# B&R Automation Studio project automationstudio
Automation Studio 4.9

## Configuration Config1

CPU X20CP1586, AutomationRuntime C4.90, Build 4.1.2, Vc V4.72.2

### Task classes (Cpu.sw)
```
Cyclic#1:
  sensors <- sensors.prg
Cyclic#3:
  main2 <- main2.prg
  main <- main.prg
Binaries: udbdef, FWRules, TCData, sysconf, Role, User, iomap, ashwd, asfw, arconfig, ashwac
Libraries: runtime, astime, asieccon, standard
```

### Hardware
```
X20CP1586 : X20CP1586 v1.8.1.0
  Connector IF2:
    ActivateDevice = 1
  ConfigurationID = sim_assigment_Config1
```

### PvMap.vvm - X20CP1586/PvMap.vvm
```iecst
VAR_CONFIG
	::robot2 AT %Q.::robot2; (*Insert your comment here...*)
	::robot1 AT %Q.::robot1; (*Insert your comment here...*)
END_VAR
```

## Logical view

Binary libraries used (declarations not repeated): standard

### Global.typ - Global data types
```iecst
TYPE
	(* Type with all sensors in scene *)
	sensorsType : STRUCT
		width : ARRAY[0..1] OF INT;
		widthBlocked : ARRAY[0..1] OF BOOL;
		height : ARRAY[0..2] OF INT;
		heightBlocked : ARRAY[0..2] OF BOOL;
		packageForPacker : BOOL;
		packageForPackerPrevious : BOOL;
	END_STRUCT;

	(* Type for holding a set from the package measuring sensors *)
	bufferType : STRUCT
		width : ARRAY[0..1] OF INT;
		height : INT;
	END_STRUCT;

	(* Type with all conveyors in scene *)
	conveyorsType : STRUCT
		circular : conveyorType;			(*  *)
		feed : conveyorType;				(*  *)
		discard : conveyorType;				(*  *)
		packer : conveyorType;				(*  *)
	END_STRUCT;
	(* Type for a specific conveyor *)
	conveyorType : STRUCT
		run : BOOL;			(*  *)
		isOn : BOOL;		(*  *)
	END_STRUCT;

	(* Singular robot control type *)
	robotType : STRUCT
		state : robotStateEnum;		(*  *)
		nextState : robotStateEnum; (*  *)
		target : robotTargetEnum;	(*  *)
		previousTarget : robotTargetEnum; (*  *)
		comm : robotCommunicationType; (*  *)
		grip : BOOL;				(*  *)
		isGripping : BOOL;			(*  *)
		inPosition : BOOL;			(*  *)
		isWaiting : BOOL;			(*  *)
	END_STRUCT;

	(* Robot state Enum *)
	robotStateEnum : (
		RSTATE_INIT, 			(*  *)
		RSTATE_FORCE_HOME,		(*  *)
		RSTATE_WAITING,		(*  *)
		RSTATE_PICKUP,		(*  *)
		RSTATE_PICKUP_R,
		RSTATE_DROP,		(*  *)
		RSTATE_DROP_R,
		RSTATE_CLEAR,
		RSTATE_E_STOP		(*  *)
	);
	(* Robot target/path Enum *)
	robotTargetEnum : (
		RTARGET_FORCE_HOME := 0,	(*  *)
		RTARGET_PICKUP_1 := 10,		(*  *)
		RTARGET_PICKUP_1_R := 11,	(*  *)
		RTARGET_PICKUP_2 := 20,		(*  *)
		RTARGET_PICKUP_2_R := 21,	(*  *)
		RTARGET_PICKUP_3 := 30,		(*  *)
		RTARGET_PICKUP_3_R := 31,	(*  *)
		RTARGET_PICKUP_4 := 40,		(*  *)
		RTARGET_PICKUP_4_R := 41,	(*  *)
		RTARGET_DROPOFF_1 := 50,	(*  *)
		RTARGET_DROPOFF_1_R := 51,	(*  *)
		RTARGET_DROPOFF_2 := 60,	(*  *)
		RTARGET_DROPOFF_2_R := 61,	(*  *)
		RTARGET_DROPOFF_3 := 70,	(*  *)
		RTARGET_DROPOFF_3_R := 71,	(*  *)
		RTARGET_CLEAR := 99			(*  *)
	);

	(*  *)
	sensorStateEnum : (
		STATE_SENSOR_CONVEYOR_INIT := 0,
		STATE_SENSOR_CONVEYOR_STOP := 1,
		STATE_SENSOR_CONVEYOR_START := 2,
		STATE_SENSOR_WAIT,
		STATE_SENSOR_MEASURING,
		STATE_SENSOR_CALCULATING,
		STATE_SENSOR_WAIT_FOR_PICKUP
	);

	(* Type for wrapping single robot comms to RobotStudio Controller *)
	robotCommunicationType : STRUCT
		targets : robotTargetType; (*  *)
		isWaiting : BOOL; (* Is waiting / ready for new action *)
		inPosition : BOOL; (* Is in the last requested position *)
		doGrip : BOOL;	(* Digital output to the gripper *)
		diGrip : BOOL; 	(* Digital input from the gripper *)
	END_STRUCT;

	(*  *)
	robotTargetType : STRUCT
		initHome : BOOL;	(* Communication to the robot *)
		home : BOOL;		(*  happens through booleans  *)
		pick1 : BOOL;		(*  only.                     *)
		pick2 : BOOL;		(* We've not been able to r/w *)
		pick3 : BOOL;		(*  other datatypes.          *)
		pick4 : BOOL;		(* initHome overrides to home *)
		drop1 : BOOL;		(* home with target reverses  *)
		drop2 : BOOL;		(*  the target path.          *)
		drop3 : BOOL;		(*                            *)
	END_STRUCT;

	(* Feeder control type *)
	packFeederType : STRUCT
		doFeed : BOOL;
		isFeeding : BOOL;
	END_STRUCT;

	(* Enum of package sizes *)
	packageSizeEnum :
		(
		PACKAGE_INVALID,
		PACKAGE_SMALL,
		PACKAGE_MEDIUM,
		PACKAGE_LARGE
	);

	(* Package type *)
	packageType : STRUCT
		width : REAL;
		length : REAL;
		height : REAL;
		volume : REAL;
		size : packageSizeEnum;	(* Package size as found after measurement *)
	END_STRUCT;

	(* Package size limit type *)
	packageSizeRangeType : STRUCT
		min : packageType;
		max : packageType;
	END_STRUCT;

	(* Accepted ranges type *)
	packingRangesType : STRUCT
		small : packageSizeRangeType;
		medium : packageSizeRangeType;
		large : packageSizeRangeType;
	END_STRUCT;

	(* Various variables used in package calculation *)
	packCalculationType : STRUCT
		cornerIndex : ARRAY[0..5] OF INT; (* Side start/end points on either side *)
		cornerIndexFilled : ARRAY[0..5] OF BOOL; (* 0..2 is for width0, 3..5 is for width1 *)
		heightIndex : ARRAY[0..1] OF INT; (* For first and second height change *)
		heightIndexFilled : ARRAY[0..1] OF BOOL; (*  *)
	END_STRUCT;
END_TYPE
```

### Global.var - Global variables
```iecst
VAR
	robot1 : robotType;	(* Robot picking from looping conveyor *)
	robot2 : robotType;	(* Robot packing onto carts *)

	sensorState : sensorStateEnum; 	(* State for sensor fsm *)

	newPack : packageType; 						(* Most recent package detected *)
	newPackR1 : packageType;				(* Current package grabbed by robot1 *)
	newPackLoaded : BOOL := FALSE;				(* Flag if robot1 has loaded newPack *)
	newPackReady : BOOL := FALSE;				(* Flag if newPack is ready for robot1 *)
	packDiscarded : BOOL := FALSE;				(* Flag is newPack has been discarded *)
	packBuffer : ARRAY[0..packBufSize] OF packageType;	(* Packs on packing conveyor *)
	packIndex : INT := 0; (* Index for the packing conveyor buffer *)
	packRanges : packingRangesType;				(* Package limits *)

	packFeeder : packFeederType;	(* Feeder control *)
	sensors : sensorsType;			(* Sensor inputs *)
	conveyors : conveyorsType;		(* Conveyor control *)

	timer_discard : TON;				(* ON timer for discard conveyor *)
	timePacking : TIME;					(* Time tracking for packing conveyor *)
	timePackingLimit : TIME := t#2s;	(* Time limit for packing conveyor *)

	packageDetectionBuffer : ARRAY[0..bufSize] OF bufferType;	(* pack sensor data buffer *)
	bufIndex : INT := 0; 		(* Index for the package detection buffer *)

	packCalc : packCalculationType; (* Struct for package size calculation *)

	Index : INT; (* Reserved for loop use *)
END_VAR

VAR CONSTANT
	LASER_DEFAULT_VALUE_HEIGHT : INT := 0;	(* No-package measurement value *)
	LASER_DEFAULT_VALUE_WIDTH : INT := 0;	(* No-package measurement value *)
	TRACK_WIDTH : INT := 650; (* Total width of the track, [mm] *)

	PACKAGE_PICKUP_LOW_LIMIT : INT := 300; (* Packages taller than this needs the high pickup *)
	PACKAGE_PICKUP_WIDTH_LIMIT : INT := 250; (* Packages with corners closer than this from right sensor gets an off-center pickup *)

	packBufSize : INT := 20 - 1; (* Elements for the packing conveyor buffer *)
	bufSize : INT := 400 - 1; (* Elements for the measurement buffer *)
END_VAR
```

### Program Logical/main (IEC)

#### Main.st
```iecst
PROGRAM _INIT
	// Package gets dropped on continuous conveyor
	// 3 laser sensors detects package size
	//		One sensor placed above to determine package height
	//		Two sensors, one either side of conveyor, to determine angle, width, and length
	// Robot1 picks up the detected package while conveyor is moving
	// If package is within an accepted range it gets put on packing conveyor
	// If package does not match, it gets discarded to an eater
	// Packages dropped to the packing conveyor gets saved in buffer
	// Robot2 picks up packages from conveyor and palletizes
	// After pickup by robot2, package is removed from buffer

	// All sensors and IO are updated in the 'sensors' loop
	// All robot1 control is done in this loop
	// All robot2 control is done in the 'main2' loop
	// Conveyors are all moving at 0.5 m/s when on

	// Package range definitions, see sensors loop
	//	Small : Volumes from 8.000.000 mm3 to 16.000.000 mm3
	//	Medium : Volumes from 16.000.000 mm3 to 32.000.000 mm3
	//	Large : Volumes from 32.000.000 to 50.000.000 mm3

	// Loop description:
	// Move to home position (close to pickup position)
	// When a package releases the sensors, newPack should be filled out by sensor loop
	// If newPack.good is true, move to packing conveyor, release, and push package to buffer
	// If newPack.good is false, move to discarding conveyor, release
	// Return to home position

	// Init the robot
	robot1.state := RSTATE_INIT;
END_PROGRAM

PROGRAM _CYCLIC

	CASE robot1.state OF
		RSTATE_INIT:
			// Set the home position target and wait for arrival
			robot1.target := RTARGET_FORCE_HOME;
			robot1.state := RSTATE_FORCE_HOME;

		RSTATE_FORCE_HOME:
			// Wait for robot to be in position
			IF robot1.inPosition THEN
				// Clear the target IO and wait
				robot1.target := RTARGET_CLEAR;
				robot1.state := RSTATE_WAITING;
			END_IF

		RSTATE_WAITING:
			// Nothing really here

		RSTATE_PICKUP:
			// Sensor loop sent us here, and set a target for us
			// Save this target
			robot1.previousTarget := robot1.target;

			// Save the package
			newPackR1 := newPack;

			// Wait for robot to be in position
			IF robot1.inPosition THEN
				// Arrived, pick up something
				robot1.grip := TRUE;
				IF robot1.isGripping THEN
					// Gripping, move back to home
					robot1.nextState := RSTATE_PICKUP_R;
					robot1.state := RSTATE_CLEAR;
				END_IF
			END_IF

		RSTATE_PICKUP_R:
			// Select reverse based on previous target
			CASE robot1.previousTarget OF
				RTARGET_PICKUP_1:
					robot1.target := RTARGET_PICKUP_1_R;

				RTARGET_PICKUP_2:
					robot1.target := RTARGET_PICKUP_2_R;

				RTARGET_PICKUP_3:
					robot1.target := RTARGET_PICKUP_3_R;

				RTARGET_PICKUP_4:
					robot1.target := RTARGET_PICKUP_4_R;

			END_CASE

			IF robot1.inPosition THEN
				// Remember some flags
				newPackLoaded := TRUE;
				newPackReady := FALSE;

				// If robot says we're home, change to drop state
				robot1.nextState := RSTATE_DROP;
				robot1.state := RSTATE_CLEAR;
			END_IF

		RSTATE_DROP:
			// Select drop target from newPackR1
			CASE newPackR1.size OF
				PACKAGE_INVALID:
					packDiscarded := TRUE;
					robot1.target := RTARGET_DROPOFF_1;

				PACKAGE_SMALL:
					robot1.target := RTARGET_DROPOFF_2;

				PACKAGE_MEDIUM:
					robot1.target := RTARGET_DROPOFF_2;

				PACKAGE_LARGE:
					robot1.target := RTARGET_DROPOFF_2;

			END_CASE

			IF robot1.target = RTARGET_DROPOFF_2 THEN
				IF packIndex < packBufSize - 1 THEN
					// Push to buffer, increment index
					packBuffer[packIndex] := newPackR1;
					packIndex := packIndex + 1;
				ELSE
					// Overflow ...
					packDiscarded := TRUE;
					robot1.target := RTARGET_DROPOFF_1;
				END_IF
			END_IF

			// Wait until we're there and the packing conveyor has moved for at least some time
			IF robot1.inPosition AND (TIME_TO_DINT(timePacking) > TIME_TO_DINT(timePackingLimit)) THEN
				// Save the target
				robot1.previousTarget := robot1.target;

				// Release the package
				robot1.grip := FALSE;
				IF NOT robot1.isGripping THEN
					// Flag
					newPackLoaded := FALSE;

					// Reset the packing conveyor timer
					timePacking := t#0s;

					// State stuff
					robot1.nextState := RSTATE_DROP_R;
					robot1.state := RSTATE_CLEAR;
				END_IF
			END_IF

		RSTATE_DROP_R:
			// Select the path home from previous target
			CASE robot1.previousTarget OF
				RTARGET_DROPOFF_1:
					robot1.target := RTARGET_DROPOFF_1_R;

				RTARGET_DROPOFF_2:
					robot1.target := RTARGET_DROPOFF_2_R;

				RTARGET_DROPOFF_3:
					robot1.target := RTARGET_DROPOFF_3_R;

			END_CASE

			// Wait for inPosition
			IF robot1.inPosition THEN
				// We're ready for new things
				robot1.state := RSTATE_CLEAR;
				robot1.nextState := RSTATE_WAITING;

			END_IF

		RSTATE_CLEAR:
			// Set the state from next set state if filled.
			// We use this to get a cycle of clear IO between moves out and back
			// Else just clear through wait
			IF NOT (robot1.nextState = RSTATE_WAITING) THEN
				robot1.state := robot1.nextState;
				robot1.target := RTARGET_CLEAR;
				robot1.previousTarget := RTARGET_CLEAR;
				robot1.nextState := RSTATE_WAITING;
			ELSE
				robot1.state := RSTATE_WAITING;
			END_IF

		RSTATE_E_STOP:
			// General kill state ..

	END_CASE

	// Write the current IO to robot comm struct, this is ugly AF
	CASE robot1.target OF
		RTARGET_FORCE_HOME:
			robot1.comm.targets.initHome := TRUE;
			robot1.comm.targets.home := FALSE;
			robot1.comm.targets.pick1 := FALSE;
			robot1.comm.targets.pick2 := FALSE;
			robot1.comm.targets.pick3 := FALSE;
			robot1.comm.targets.pick4 := FALSE;
			robot1.comm.targets.drop1 := FALSE;
			robot1.comm.targets.drop2 := FALSE;
			robot1.comm.targets.drop3 := FALSE;

		RTARGET_PICKUP_1:
			robot1.comm.targets.initHome := FALSE;
			robot1.comm.targets.home := FALSE;
			robot1.comm.targets.pick1 := TRUE;
			robot1.comm.targets.pick2 := FALSE;
			robot1.comm.targets.pick3 := FALSE;
			robot1.comm.targets.pick4 := FALSE;
			robot1.comm.targets.drop1 := FALSE;
			robot1.comm.targets.drop2 := FALSE;
			robot1.comm.targets.drop3 := FALSE;
		RTARGET_PICKUP_1_R:
			robot1.comm.targets.initHome := FALSE;
			robot1.comm.targets.home := TRUE;
			robot1.comm.targets.pick1 := TRUE;
			robot1.comm.targets.pick2 := FALSE;
			robot1.comm.targets.pick3 := FALSE;
			robot1.comm.targets.pick4 := FALSE;
			robot1.comm.targets.drop1 := FALSE;
			robot1.comm.targets.drop2 := FALSE;
			robot1.comm.targets.drop3 := FALSE;

		RTARGET_PICKUP_2:
			robot1.comm.targets.initHome := FALSE;
			robot1.comm.targets.home := FALSE;
			robot1.comm.targets.pick1 := FALSE;
			robot1.comm.targets.pick2 := TRUE;
			robot1.comm.targets.pick3 := FALSE;
			robot1.comm.targets.pick4 := FALSE;
			robot1.comm.targets.drop1 := FALSE;
			robot1.comm.targets.drop2 := FALSE;
			robot1.comm.targets.drop3 := FALSE;
		RTARGET_PICKUP_2_R:
			robot1.comm.targets.initHome := FALSE;
			robot1.comm.targets.home := TRUE;
			robot1.comm.targets.pick1 := FALSE;
			robot1.comm.targets.pick2 := TRUE;
			robot1.comm.targets.pick3 := FALSE;
			robot1.comm.targets.pick4 := FALSE;
			robot1.comm.targets.drop1 := FALSE;
			robot1.comm.targets.drop2 := FALSE;
			robot1.comm.targets.drop3 := FALSE;

		RTARGET_PICKUP_3:
			robot1.comm.targets.initHome := FALSE;
			robot1.comm.targets.home := FALSE;
			robot1.comm.targets.pick1 := FALSE;
			robot1.comm.targets.pick2 := FALSE;
			robot1.comm.targets.pick3 := TRUE;
			robot1.comm.targets.pick4 := FALSE;
			robot1.comm.targets.drop1 := FALSE;
			robot1.comm.targets.drop2 := FALSE;
			robot1.comm.targets.drop3 := FALSE;
		RTARGET_PICKUP_3_R:
			robot1.comm.targets.initHome := FALSE;
			robot1.comm.targets.home := TRUE;
			robot1.comm.targets.pick1 := FALSE;
			robot1.comm.targets.pick2 := FALSE;
			robot1.comm.targets.pick3 := TRUE;
			robot1.comm.targets.pick4 := FALSE;
			robot1.comm.targets.drop1 := FALSE;
			robot1.comm.targets.drop2 := FALSE;
			robot1.comm.targets.drop3 := FALSE;

		RTARGET_PICKUP_4:
			robot1.comm.targets.initHome := FALSE;
			robot1.comm.targets.home := FALSE;
			robot1.comm.targets.pick1 := FALSE;
			robot1.comm.targets.pick2 := FALSE;
			robot1.comm.targets.pick3 := FALSE;
			robot1.comm.targets.pick4 := TRUE;
			robot1.comm.targets.drop1 := FALSE;
			robot1.comm.targets.drop2 := FALSE;
			robot1.comm.targets.drop3 := FALSE;
		RTARGET_PICKUP_4_R:
			robot1.comm.targets.initHome := FALSE;
			robot1.comm.targets.home := TRUE;
			robot1.comm.targets.pick1 := FALSE;
			robot1.comm.targets.pick2 := FALSE;
			robot1.comm.targets.pick3 := FALSE;
			robot1.comm.targets.pick4 := TRUE;
			robot1.comm.targets.drop1 := FALSE;
			robot1.comm.targets.drop2 := FALSE;
			robot1.comm.targets.drop3 := FALSE;

		RTARGET_DROPOFF_1:
			robot1.comm.targets.initHome := FALSE;
			robot1.comm.targets.home := FALSE;
			robot1.comm.targets.pick1 := FALSE;
			robot1.comm.targets.pick2 := FALSE;
			robot1.comm.targets.pick3 := FALSE;
			robot1.comm.targets.pick4 := FALSE;
			robot1.comm.targets.drop1 := TRUE;
			robot1.comm.targets.drop2 := FALSE;
			robot1.comm.targets.drop3 := FALSE;
		RTARGET_DROPOFF_1_R:
			robot1.comm.targets.initHome := FALSE;
			robot1.comm.targets.home := TRUE;
			robot1.comm.targets.pick1 := FALSE;
			robot1.comm.targets.pick2 := FALSE;
			robot1.comm.targets.pick3 := FALSE;
			robot1.comm.targets.pick4 := FALSE;
			robot1.comm.targets.drop1 := TRUE;
			robot1.comm.targets.drop2 := FALSE;
			robot1.comm.targets.drop3 := FALSE;

		RTARGET_DROPOFF_2:
			robot1.comm.targets.initHome := FALSE;
			robot1.comm.targets.home := FALSE;
			robot1.comm.targets.pick1 := FALSE;
			robot1.comm.targets.pick2 := FALSE;
			robot1.comm.targets.pick3 := FALSE;
			robot1.comm.targets.pick4 := FALSE;
			robot1.comm.targets.drop1 := FALSE;
			robot1.comm.targets.drop2 := TRUE;
			robot1.comm.targets.drop3 := FALSE;
		RTARGET_DROPOFF_2_R:
			robot1.comm.targets.initHome := FALSE;
			robot1.comm.targets.home := TRUE;
			robot1.comm.targets.pick1 := FALSE;
			robot1.comm.targets.pick2 := FALSE;
			robot1.comm.targets.pick3 := FALSE;
			robot1.comm.targets.pick4 := FALSE;
			robot1.comm.targets.drop1 := FALSE;
			robot1.comm.targets.drop2 := TRUE;
			robot1.comm.targets.drop3 := FALSE;

		RTARGET_DROPOFF_3:
			robot1.comm.targets.initHome := FALSE;
			robot1.comm.targets.home := FALSE;
			robot1.comm.targets.pick1 := FALSE;
			robot1.comm.targets.pick2 := FALSE;
			robot1.comm.targets.pick3 := FALSE;
			robot1.comm.targets.pick4 := FALSE;
			robot1.comm.targets.drop1 := FALSE;
			robot1.comm.targets.drop2 := FALSE;
			robot1.comm.targets.drop3 := TRUE;
		RTARGET_DROPOFF_3_R:
			robot1.comm.targets.initHome := FALSE;
			robot1.comm.targets.home := TRUE;
			robot1.comm.targets.pick1 := FALSE;
			robot1.comm.targets.pick2 := FALSE;
			robot1.comm.targets.pick3 := FALSE;
			robot1.comm.targets.pick4 := FALSE;
			robot1.comm.targets.drop1 := FALSE;
			robot1.comm.targets.drop2 := FALSE;
			robot1.comm.targets.drop3 := TRUE;

		RTARGET_CLEAR:
			robot1.comm.targets.initHome := FALSE;
			robot1.comm.targets.home := FALSE;
			robot1.comm.targets.pick1 := FALSE;
			robot1.comm.targets.pick2 := FALSE;
			robot1.comm.targets.pick3 := FALSE;
			robot1.comm.targets.pick4 := FALSE;
			robot1.comm.targets.drop1 := FALSE;
			robot1.comm.targets.drop2 := FALSE;
			robot1.comm.targets.drop3 := FALSE;

	END_CASE
	robot1.comm.doGrip := robot1.grip;
	robot1.isGripping := robot1.comm.diGrip;
	robot1.inPosition := robot1.comm.inPosition;
	robot1.isWaiting := robot1.comm.isWaiting;

END_PROGRAM

PROGRAM _EXIT

END_PROGRAM
```

### Program Logical/sensors (IEC)

#### Main.st
```iecst
PROGRAM _INIT
	// Loop description

	// SENSORS ON THE CIRCULAR CONVEYOR
	// When a new package is detected, start recording measurements
	// When package releases, calculate angle and actual size / volume
		// If robot1 is currently away from waiting position, pause the conveyor or ignore the package
	// Fill result into newPack and determine if it is 'good'
	// If new package is detected before newPackLoaded is true, stop the feeder and conveyor
	// If no gap is detected between two packages, ignore the second package

	// SENSOR ON THE PACKING CONVEYOR
	// If sensor is activated, stop the conveyor until it is de-activated again

	// Lasers in Experior are very very broken
	// They cannot do distance measurements unless perfectly level
	// This was only found out after preparing for it..

	// Initializing the accepted package sizes
	packRanges.small.min.volume := 8000000; 				(*  8.000.000 mm3 *)
	packRanges.small.max.volume := 16000000; 				(* 16.000.000 mm3 *)
	packRanges.medium.min.volume := packRanges.small.max.volume;
	packRanges.medium.max.volume := 32000000;				(* 32.000.000 mm3 *)
	packRanges.large.min.volume := packRanges.medium.max.volume;
	packRanges.large.max.volume := 50000000;				(* 50.000.000 mm3 *)

	// Initialize the timer
	timer_discard.PT := t#3s;
END_PROGRAM

PROGRAM _CYCLIC
	// Conveyor fsm
	CASE sensorState OF
		STATE_SENSOR_CONVEYOR_INIT:
			// Restart the tracks, Experior doesn't read on connection properly?
			conveyors.circular.run := TRUE;
			conveyors.discard.run := TRUE;
			conveyors.feed.run := TRUE;
			conveyors.packer.run := TRUE;
			sensorState := STATE_SENSOR_CONVEYOR_STOP;

		STATE_SENSOR_CONVEYOR_STOP:
			// Restart the tracks, Experior doesn't read on connection properly?
			conveyors.circular.run := FALSE;
			conveyors.discard.run := FALSE;
			conveyors.feed.run := FALSE;
			conveyors.packer.run := FALSE;
			sensorState := STATE_SENSOR_CONVEYOR_START;

		STATE_SENSOR_CONVEYOR_START:
			// Start them again and check
			conveyors.circular.run := TRUE;
			conveyors.discard.run := TRUE;
			conveyors.feed.run := TRUE;
			conveyors.packer.run := TRUE;

			//// Experior doesn't really like updating the inputs, so we'll be ignoring them ..
			//IF conveyors.circular.isOn AND conveyors.discard.isOn AND conveyors.feed.isOn AND conveyors.packer.isOn THEN
				// Change state if both robots are also ready

				IF robot1.state = RSTATE_WAITING AND robot2.state = RSTATE_WAITING THEN
					packFeeder.doFeed := TRUE;
					sensorState := STATE_SENSOR_MEASURING;
				END_IF

			//END_IF

		STATE_SENSOR_WAIT:
			IF sensors.widthBlocked[0] OR sensors.widthBlocked[1] THEN
				// Reset buffer index
				bufIndex := 0;

				// Grab first set of data
				//packageDetectionBuffer[bufIndex].height := MAX(sensors.height[0], sensors.height[1], sensors.height[2]);
				packageDetectionBuffer[bufIndex].height := 300; (* Let's pretend it's always 300mm. I blame Experior. *)
				packageDetectionBuffer[bufIndex].width := sensors.width;

				// Increment index
				bufIndex := bufIndex + 1;

				// Change to continuos measuring state
				sensorState := STATE_SENSOR_MEASURING;
			END_IF

		STATE_SENSOR_MEASURING:
			// When a package is detected, save first set of data and enter continuous measurement
			IF sensors.widthBlocked[0] OR sensors.widthBlocked[1] THEN
				// Grab a set of data while either sensor is still blocked
				//packageDetectionBuffer[bufIndex].height := MAX(sensors.height[0], sensors.height[1], sensors.height[2]);
				packageDetectionBuffer[bufIndex].height := 300; (* Let's pretend it's always 300mm. I blame Experior. *)
				packageDetectionBuffer[bufIndex].width := sensors.width;

				// Increment the buffer index
				IF bufIndex > bufSize - 1 THEN
					// Size overflow, just change to the next state
					sensorState := STATE_SENSOR_CALCULATING;
				ELSE
					// Increment for next measurement
					bufIndex := bufIndex + 1;
				END_IF
			ELSE
				// Change to the calculation state
				sensorState := STATE_SENSOR_CALCULATING;
			END_IF

		STATE_SENSOR_CALCULATING:
			// Stop the tracks, robot1 isn't happy about them moving while picking up
			conveyors.circular.run := FALSE;
			conveyors.feed.run := FALSE;

			// Find the package stuff, prime robot1 and the required track for movement
			// We assume a box shape. BufIndex isn't a filled value.
			// Find a corner
			FOR Index:=0 TO bufIndex - 2 DO

				// Resolution in the track direction isn't great, 0.5 m/s @ 10ms samples = 5mm
				// Also the Laser sensors in Experior are very unreliable in general ...

				//// Width sensor 0
				IF NOT (packageDetectionBuffer[Index].width[0] = LASER_DEFAULT_VALUE_WIDTH) THEN
					// Valid measurement
					// Save initial detection position in packCalc
					IF NOT packCalc.cornerIndexFilled[0] THEN
						packCalc.cornerIndex[0] := Index;
						packCalc.cornerIndexFilled[0] := TRUE;
					END_IF
					// Sensors will always start going down, as free measurement is high limit
					// If box is square on, they will not change
					// If box is angled, it will ramp up until a corner, and ramp back down after.
					// Some detector measurement error has to be allowable, as a false positive wrecks the "algorithm"
					// However this is simulated, so we won't
					IF packageDetectionBuffer[Index].width[0] < packageDetectionBuffer[Index + 1].width[0] THEN
						// Corner found
						IF NOT packCalc.cornerIndexFilled[1] THEN
							packCalc.cornerIndex[1] := Index;
							packCalc.cornerIndexFilled[1] := TRUE;
						END_IF
					END_IF
					// Check for a ramp going up after finding the corner, that would be a new box
					IF packageDetectionBuffer[Index].width[0] > packageDetectionBuffer[Index + 1].width[0] AND packCalc.cornerIndexFilled[1] THEN
						IF NOT packCalc.cornerIndexFilled[2] THEN
							packCalc.cornerIndex[2] := Index;
							packCalc.cornerIndexFilled[2] := TRUE;
						END_IF
					END_IF
				ELSIF packCalc.cornerIndexFilled[0] AND NOT packCalc.cornerIndexFilled[2] THEN
					// If sensor is free and we did find the first point, this is the end
					// If the third point is already filled, we found another box instead
					// We decrement the index to save the last valid measurement instead of the first invalid one
					packCalc.cornerIndex[2] := Index - 1;
					packCalc.cornerIndexFilled[2] := TRUE;
				END_IF

				//// Width sensor 1 (copied from width sensor 0)
				IF NOT packageDetectionBuffer[Index].width[1] = LASER_DEFAULT_VALUE_WIDTH THEN
					// Valid measurement
					// Save initial detection position in packCalc
					IF NOT packCalc.cornerIndexFilled[3] THEN
						packCalc.cornerIndex[3] := Index;
						packCalc.cornerIndexFilled[3] := TRUE;
					END_IF
					// Sensors will always start going down, as free measurement is high limit
					// If box is square on, they will not change
					// If box is angled, it will ramp up until a corner, and ramp back down after.
					// Some detector measurement error has to be allowable, as a false positive wrecks the "algorithm"
					// However this is simulated, so we won't
					IF packageDetectionBuffer[Index].width[1] < packageDetectionBuffer[Index + 1].width[1] THEN
						// Corner found
						IF NOT packCalc.cornerIndexFilled[4] THEN
							packCalc.cornerIndex[4] := Index;
							packCalc.cornerIndexFilled[4] := TRUE;
						END_IF
					END_IF
					// Check for a ramp going up after finding the corner, that would be a new box
					IF packageDetectionBuffer[Index].width[1] > packageDetectionBuffer[Index + 1].width[1] AND packCalc.cornerIndexFilled[4] THEN
						IF NOT packCalc.cornerIndexFilled[5] THEN
							packCalc.cornerIndex[5] := Index;
							packCalc.cornerIndexFilled[5] := TRUE;
						END_IF
					END_IF
				ELSIF packCalc.cornerIndexFilled[3] AND NOT packCalc.cornerIndexFilled[5] THEN
					// If sensor is free and we did find the first point, this is the end
					// If the third point is already filled, we found another box instead
					// We decrement the index to save the last valid measurement instead of the first invalid one
					packCalc.cornerIndex[5] := Index - 1;
					packCalc.cornerIndexFilled[5] := TRUE;
				END_IF
			END_FOR

			// Finding the dimensions
			IF packCalc.cornerIndexFilled[0] AND packCalc.cornerIndexFilled[1] AND packCalc.cornerIndexFilled[2] AND
				packCalc.cornerIndexFilled[3] AND packCalc.cornerIndexFilled[4] AND packCalc.cornerIndexFilled[5] THEN
				// All corners detected
				// Width of box: sqrt ( (dx)^2 + (dy)^2 )
				// dx = trackwidth - sensor distance at mid corner - sensor distance at trailing corner
				// dy = track velocity * cycles spent from mid corner to trailing corner * cycle time
				newPack.width := SQRT(
				(TRACK_WIDTH - packageDetectionBuffer[packCalc.cornerIndex[1]].width[0] - packageDetectionBuffer[packCalc.cornerIndex[2]].width[1])
				* (TRACK_WIDTH - packageDetectionBuffer[packCalc.cornerIndex[1]].width[0] - packageDetectionBuffer[packCalc.cornerIndex[2]].width[1])
				+ (0.5 * (packCalc.cornerIndex[2] - packCalc.cornerIndex[1]) * 10)
				* (0.5 * (packCalc.cornerIndex[2] - packCalc.cornerIndex[1]) * 10)
				);

				// Length is found in a similar fashion
				newPack.width := SQRT(
				(TRACK_WIDTH - packageDetectionBuffer[packCalc.cornerIndex[4]].width[1] - packageDetectionBuffer[packCalc.cornerIndex[2]].width[0])
				* (TRACK_WIDTH - packageDetectionBuffer[packCalc.cornerIndex[4]].width[1] - packageDetectionBuffer[packCalc.cornerIndex[2]].width[0])
				+ (0.5 * (packCalc.cornerIndex[2] - packCalc.cornerIndex[4]) * 10)
				* (0.5 * (packCalc.cornerIndex[2] - packCalc.cornerIndex[4]) * 10)
				);

				// Height is taken at the mid-corner point
				newPack.height := LASER_DEFAULT_VALUE_HEIGHT - packageDetectionBuffer[packCalc.cornerIndex[1]].height;

			ELSIF packCalc.cornerIndexFilled[0] AND NOT packCalc.cornerIndexFilled[1] AND packCalc.cornerIndexFilled[2] AND
				packCalc.cornerIndexFilled[3] AND NOT packCalc.cornerIndexFilled[4] AND packCalc.cornerIndexFilled[5] THEN
				// Midpoint(s) not found, randomly perfectly straight box?
				// Makes it easy enough
				newPack.width := TRACK_WIDTH - packageDetectionBuffer[REAL_TO_INT((packCalc.cornerIndex[0] + packCalc.cornerIndex[2]) / 2)].width[0] - packageDetectionBuffer[REAL_TO_INT((packCalc.cornerIndex[0] + packCalc.cornerIndex[2]) / 2)].width[1];
				newPack.height := 300; (* The laser in Experior doesn't want to work in vertical orientation .. *)
				newPack.length := 0.5 * (packCalc.cornerIndex[2] - packCalc.cornerIndex[0]) * 10;
			END_IF

			// Calculate volume from found WxLxH and select the package size type
			newPack.volume := newPack.height * newPack.width * newPack.length;
			IF newPack.volume >= packRanges.small.min.volume AND newPack.volume <= packRanges.small.max.volume THEN
				// Pack is inside the 'small' range
				newPack.size := PACKAGE_SMALL;
			ELSIF newPack.volume >= packRanges.medium.min.volume AND newPack.volume <= packRanges.medium.max.volume THEN
				// Pack is inside the 'medium' range
				newPack.size := PACKAGE_MEDIUM;
			ELSIF newPack.volume >= packRanges.large.min.volume AND newPack.volume <= packRanges.large.max.volume THEN
				// Pack is inside the 'large' range
				newPack.size := PACKAGE_LARGE;
			ELSE
				// Pack not in any ranges;
				newPack.size := PACKAGE_INVALID;
			END_IF

			// Reset the flag for new package to be loaded by robot1
			newPackReady := TRUE;

			// Set robot1 target position based on package height and position on track
			IF packageDetectionBuffer[packCalc.cornerIndex[1]].height > PACKAGE_PICKUP_LOW_LIMIT THEN
				IF packageDetectionBuffer[packCalc.cornerIndex[1]].width[0] > PACKAGE_PICKUP_WIDTH_LIMIT THEN
					robot1.target := RTARGET_PICKUP_1;
				ELSE
					robot1.target := RTARGET_PICKUP_2;
				END_IF
			ELSE
				IF packageDetectionBuffer[packCalc.cornerIndex[1]].width[0] > PACKAGE_PICKUP_WIDTH_LIMIT THEN
					robot1.target := RTARGET_PICKUP_3;
				ELSE
					robot1.target := RTARGET_PICKUP_4;
				END_IF
			END_IF

			// Start robot1 via the pickup state
			robot1.state := RSTATE_PICKUP;

			// Reset the buffer index to pseudo clear it
			bufIndex := 0;

			// Clear the packCalc
			FOR Index:=0 TO 5 DO
				packCalc.cornerIndex[Index] := FALSE;
				packCalc.cornerIndexFilled[Index] := FALSE;
			END_FOR
			FOR Index:=0 TO 1 DO
				packCalc.heightIndex[Index] := FALSE;
				packCalc.heightIndexFilled[Index] := FALSE;
			END_FOR

			// Change the sensor loop state
			sensorState := STATE_SENSOR_WAIT_FOR_PICKUP;

		STATE_SENSOR_WAIT_FOR_PICKUP:
			// Wait until robot1 has picked up the package
			IF NOT newPackReady THEN
				// Package has been cleared by the robot, restart the conveyors and feeder
				conveyors.circular.run := TRUE;
				conveyors.feed.run := TRUE;
				packFeeder.doFeed := TRUE;

				// Change to the waiting state
				sensorState := STATE_SENSOR_WAIT_FOR_PICKUP;
			END_IF
	END_CASE

	//////////////////////////
	// This is an old block of code
	//////////////////////////

//	// Conveyor loop
//	// Measuring packages if sensors show anything on width
//	IF (sensors.widthBlocked[0] OR
//		sensors.widthBlocked[1]) AND
//		NOT doublePackageDetected THEN
//
//		// Set the 'currently measuring' flag
//		packageInDetection := TRUE;
//
//		// Lasers in Experior are very very broken
//		// They cannot do distance measurements unless perfectly level
//		// This was only found out after preparing for it..
//
//		// Grab a set of data
//		//packageDetectionBuffer[bufIndex].height := MAX(sensors.height[0], sensors.height[1], sensors.height[2]);
//		packageDetectionBuffer[bufIndex].height := 300; (* Let's pretend it's always 300mm. I blame Experior. *)
//		packageDetectionBuffer[bufIndex].width := sensors.width;
//
//		// TODO: Do a check to see if we have transitioned to measuring a new package?
//		// Check if width has changed direction twice??
//		// Move to next step by using "doublePackageDetected" and ignore the second package
//		// Maybe some check to stop the feeder if conveyor is filled?
//
//		// Increment the buffer index, and check for overflow
//		IF bufIndex > bufSize - 1 THEN
//			// Size overflow, just set the flag for multiple packages
//			doublePackageDetected := TRUE;
//		ELSE
//			// Increment for next measurement
//			bufIndex := bufIndex + 1;
//		END_IF
//
//	ELSIF packageInDetection OR doublePackageDetected THEN
//		// Sensors didn't detect anything after measuring, or second pack is detected
//		// Reset the flags
//		packageInDetection := FALSE;
//		doublePackageDetected := FALSE;
//
//		// If the newPackLoaded it true and robot1 is ready for pickup, fill newPack and start robot1
//		// If not, ignore the package. The robot might not be able to reach it in time
//		// TODO: Somehow check if the circular conveyor is overfilled?
//		IF newPackLoaded AND robot1.state = RSTATE_WAITING THEN
//			// We assume a box shape. BufIndex should be a filled measurement.
//			// Find a corner
//			FOR Index:=0 TO bufIndex - 1 DO
//
//				// Resolution in the track direction isn't great, 0.5 m/s @ 10ms samples = 5mm
//
//				//// Width sensor 0
//				IF NOT packageDetectionBuffer[Index].width[0] = LASER_DEFAULT_VALUE_WIDTH THEN
//					// Valid measurement
//					// Save initial detection position in packCalc
//					IF NOT packCalc.cornerIndexFilled[0] THEN
//						packCalc.cornerIndex[0] := Index;
//						packCalc.cornerIndexFilled[0] := TRUE;
//					END_IF
//					// Sensors will always start going down, as free measurement is high limit
//					// If box is square on, they will not change
//					// If box is angled, it will ramp up until a corner, and ramp back down after.
//					// Some detector measurement error has to be allowable, as a false positive wrecks the "algorithm"
//					// However this is simulated, so we won't
//					IF packageDetectionBuffer[Index].width[0] < packageDetectionBuffer[Index + 1].width[0] THEN
//						// Corner found
//						IF NOT packCalc.cornerIndexFilled[1] THEN
//							packCalc.cornerIndex[1] := Index;
//							packCalc.cornerIndexFilled[1] := TRUE;
//						END_IF
//					END_IF
//					// Check for a ramp going up after finding the corner, that would be a new box
//					IF packageDetectionBuffer[Index].width[0] > packageDetectionBuffer[Index + 1].width[0] AND packCalc.cornerIndexFilled[1] THEN
//						IF NOT packCalc.cornerIndexFilled[2] THEN
//							packCalc.cornerIndex[2] := Index;
//							packCalc.cornerIndexFilled[2] := TRUE;
//						END_IF
//					END_IF
//				ELSIF packCalc.cornerIndexFilled[0] AND NOT packCalc.cornerIndexFilled[2] THEN
//					// If sensor is free and we did find the first point, this is the end
//					// If the third point is already filled, we found another box instead
//					// We decrement the index to save the last valid measurement instead of the first invalid one
//					packCalc.cornerIndex[2] := Index - 1;
//					packCalc.cornerIndexFilled[2] := TRUE;
//				END_IF
//
//				//// Width sensor 1 (copied from width sensor 0)
//				IF NOT packageDetectionBuffer[Index].width[1] = LASER_DEFAULT_VALUE_WIDTH THEN
//					// Valid measurement
//					// Save initial detection position in packCalc
//					IF NOT packCalc.cornerIndexFilled[3] THEN
//						packCalc.cornerIndex[3] := Index;
//						packCalc.cornerIndexFilled[3] := TRUE;
//					END_IF
//					// Sensors will always start going down, as free measurement is high limit
//					// If box is square on, they will not change
//					// If box is angled, it will ramp up until a corner, and ramp back down after.
//					// Some detector measurement error has to be allowable, as a false positive wrecks the "algorithm"
//					// However this is simulated, so we won't
//					IF packageDetectionBuffer[Index].width[1] < packageDetectionBuffer[Index + 1].width[1] THEN
//						// Corner found
//						IF NOT packCalc.cornerIndexFilled[4] THEN
//							packCalc.cornerIndex[4] := Index;
//							packCalc.cornerIndexFilled[4] := TRUE;
//						END_IF
//					END_IF
//					// Check for a ramp going up after finding the corner, that would be a new box
//					IF packageDetectionBuffer[Index].width[1] > packageDetectionBuffer[Index + 1].width[1] AND packCalc.cornerIndexFilled[4] THEN
//						IF NOT packCalc.cornerIndexFilled[5] THEN
//							packCalc.cornerIndex[5] := Index;
//							packCalc.cornerIndexFilled[5] := TRUE;
//						END_IF
//					END_IF
//				ELSIF packCalc.cornerIndexFilled[3] AND NOT packCalc.cornerIndexFilled[5] THEN
//					// If sensor is free and we did find the first point, this is the end
//					// If the third point is already filled, we found another box instead
//					// We decrement the index to save the last valid measurement instead of the first invalid one
//					packCalc.cornerIndex[5] := Index - 1;
//					packCalc.cornerIndexFilled[5] := TRUE;
//				END_IF
//			END_FOR
//
//			// For finding the dimensions, lets find the distance measured on the middle of each side
//			IF packCalc.cornerIndexFilled[0] AND packCalc.cornerIndexFilled[1] AND packCalc.cornerIndexFilled[2] AND
//				packCalc.cornerIndexFilled[3] AND packCalc.cornerIndexFilled[4] AND packCalc.cornerIndexFilled[5] THEN
//				// All corners detected
//				packCalc.sideMidPoint[0] := REAL_TO_INT(0.5 * INT_TO_REAL(packCalc.cornerIndex[0] + packCalc.cornerIndex[1]));
//				packCalc.sideMidPoint[1] := REAL_TO_INT(0.5 * INT_TO_REAL(packCalc.cornerIndex[1] + packCalc.cornerIndex[2]));
//				packCalc.sideMidPoint[2] := REAL_TO_INT(0.5 * INT_TO_REAL(packCalc.cornerIndex[3] + packCalc.cornerIndex[4]));
//				packCalc.sideMidPoint[3] := REAL_TO_INT(0.5 * INT_TO_REAL(packCalc.cornerIndex[4] + packCalc.cornerIndex[5]));
//
//				// Width of box: sqrt ( (dx)^2 + (dy)^2 )
//				// dx = trackwidth - sensor distance at mid corner - sensor distance at trailing corner
//				// dy = track velocity * cycles spent from mid corner to trailing corner * cycle time
//				newPack.width := SQRT(
//					(TRACK_WIDTH - packageDetectionBuffer[packCalc.cornerIndex[1]].width[0] - packageDetectionBuffer[packCalc.cornerIndex[2]].width[1])
//					* (TRACK_WIDTH - packageDetectionBuffer[packCalc.cornerIndex[1]].width[0] - packageDetectionBuffer[packCalc.cornerIndex[2]].width[1])
//					+ (0.5 * (packCalc.cornerIndex[2] - packCalc.cornerIndex[1]) * 10)
//					* (0.5 * (packCalc.cornerIndex[2] - packCalc.cornerIndex[1]) * 10)
//				);
//
//				// Length is found in a similar fashion
//				newPack.width := SQRT(
//					(TRACK_WIDTH - packageDetectionBuffer[packCalc.cornerIndex[4]].width[1] - packageDetectionBuffer[packCalc.cornerIndex[2]].width[0])
//					* (TRACK_WIDTH - packageDetectionBuffer[packCalc.cornerIndex[4]].width[1] - packageDetectionBuffer[packCalc.cornerIndex[2]].width[0])
//					+ (0.5 * (packCalc.cornerIndex[2] - packCalc.cornerIndex[4]) * 10)
//					* (0.5 * (packCalc.cornerIndex[2] - packCalc.cornerIndex[4]) * 10)
//				);
//
//				// Height is taken at the mid-corner point
//				newPack.height := LASER_DEFAULT_VALUE_HEIGHT - packageDetectionBuffer[packCalc.cornerIndex[1]].height;
//
//
//			ELSIF packCalc.cornerIndexFilled[0] AND NOT packCalc.cornerIndexFilled[1] AND packCalc.cornerIndexFilled[2] AND
//				packCalc.cornerIndexFilled[3] AND NOT packCalc.cornerIndexFilled[4] AND packCalc.cornerIndexFilled[5] THEN
//				// Midpoint(s) not found, randomly perfectly straight box?
//				// Makes it easy enough
//				packCalc.sideMidPoint[0] := REAL_TO_INT(0.5 * INT_TO_REAL(packCalc.cornerIndex[0] + packCalc.cornerIndex[2]));
//
//				newPack.width := TRACK_WIDTH - packageDetectionBuffer[packCalc.sideMidPoint[0]].width[0] - packageDetectionBuffer[packCalc.sideMidPoint[0]].width[1];
//				newPack.height := LASER_DEFAULT_VALUE_HEIGHT - packageDetectionBuffer[packCalc.sideMidPoint[0]].height;
//				newPack.length := 0.5 * (packCalc.cornerIndex[2] - packCalc.cornerIndex[0]) * 10;
//			END_IF
//
//			// Calculate volume from found WxLxH and select the package size type
//			newPack.volume := newPack.height * newPack.width * newPack.length;
//			IF newPack.volume >= packRanges.small.min.volume AND newPack.volume <= packRanges.small.max.volume THEN
//				// Pack is inside the 'small' range
//				newPack.size := PACKAGE_SMALL;
//			ELSIF newPack.volume >= packRanges.medium.min.volume AND newPack.volume <= packRanges.medium.max.volume THEN
//				// Pack is inside the 'medium' range
//				newPack.size := PACKAGE_MEDIUM;
//			ELSIF newPack.volume >= packRanges.large.min.volume AND newPack.volume <= packRanges.large.max.volume THEN
//				// Pack is inside the 'large' range
//				newPack.size := PACKAGE_LARGE;
//			ELSE
//				// Pack not in any ranges;
//				newPack.size := PACKAGE_INVALID;
//			END_IF
//
//			// Reset the flag for new package to be loaded by robot1
//			newPackReady := TRUE;
//
//			// Set robot1 target position based on package height and position on track
//			IF packageDetectionBuffer[packCalc.cornerIndex[1]].height > PACKAGE_PICKUP_LOW_LIMIT THEN
//				IF packageDetectionBuffer[packCalc.cornerIndex[1]].width[0] > PACKAGE_PICKUP_WIDTH_LIMIT THEN
//					robot1.target := RTARGET_PICKUP_1;
//				ELSE
//					robot1.target := RTARGET_PICKUP_2;
//				END_IF
//			ELSE
//				IF packageDetectionBuffer[packCalc.cornerIndex[1]].width[0] > PACKAGE_PICKUP_WIDTH_LIMIT THEN
//					robot1.target := RTARGET_PICKUP_3;
//				ELSE
//					robot1.target := RTARGET_PICKUP_4;
//				END_IF
//			END_IF
//
//			// Start robot1 via the pickup state
//			robot1.state := RSTATE_PICKUP;
//
//		END_IF
//
//		// Pseudo-clear the buffer by resetting the index
//		bufIndex := 0;
//
//	END_IF

	// Circular conveyor
//	IF newPackReady AND (robot1.state = RSTATE_WAITING OR robot1.state = RSTATE_PICKUP) THEN
//		// We can only pick up stationary packages, so wait for robot1 to clear the package
//		conveyors.circular := FALSE;
//		// Also stop the package feeder
//		packFeeder.doFeed := FALSE;
//	ELSIF newPackLoaded THEN
//		// Start the conveyor when a pack is done being grabbed
//		conveyors.circular := TRUE;
//		packFeeder.doFeed := TRUE;
//	END_IF

	//////////////////////////
	// This is the end of an old block of code
	//////////////////////////

	// Packing conveyor
	IF sensors.packageForPacker THEN
		// Stop the conveyor
		conveyors.packer.run := FALSE;
		// Start pickup once robot is ready
		IF robot2.state = RSTATE_WAITING THEN
			// Low packages get a lower pickup point
			IF packBuffer[0].height > PACKAGE_PICKUP_LOW_LIMIT THEN
				robot2.target := RTARGET_PICKUP_1;
			ELSE
				robot2.target := RTARGET_PICKUP_2;
			END_IF
			robot2.state := RSTATE_PICKUP;
		END_IF
	ELSE
		// If the above fsm is in state 3 or higher, just force the packer high
		IF sensorState > 2 THEN
			conveyors.packer.run := TRUE;
		END_IF

		// Update time spent moving since drop
		// robot1 checks for this time to exceed a value in the main loop
		IF conveyors.packer.isOn THEN
			timePacking := timePacking + t#10ms;
		END_IF

		// If first time here since last activation, pop a package from buffer by shifting them
		IF sensors.packageForPackerPrevious THEN
			sensors.packageForPackerPrevious := sensors.packageForPacker;
			FOR Index:=0 TO packBufSize - 1 DO
				packBuffer[Index] := packBuffer[Index + 1];
			END_FOR
		END_IF

	END_IF

	// Discarding conveyor
	IF packDiscarded THEN
		// Reset flag
		packDiscarded := FALSE;

		// Run conveyor
		conveyors.discard.run := TRUE;

		// If timer is already running, hard reset
		IF timer_discard.IN THEN
			timer_discard.IN := FALSE;
			timer_discard();
		END_IF

		// Start the timer
		timer_discard.IN := TRUE;

	ELSIF timer_discard.Q THEN
		// Stop the timer when done
		timer_discard.IN := FALSE;

		// Stop the conveyor
		conveyors.discard.run := FALSE;
	END_IF

	// Update the timer block for discard conveyor
	timer_discard();

	// Feed conveyor gets the same state as the circular one
	conveyors.feed.run := conveyors.circular.run;

END_PROGRAM

PROGRAM _EXIT
	// Stop all of the things we can
	// Probably useless since we're dying fast

	conveyors.circular.run := FALSE;
	conveyors.discard.run := FALSE;
	conveyors.packer.run := FALSE;
	conveyors.feed.run := FALSE;
	robot1.state := RSTATE_E_STOP;
	robot2.state := RSTATE_E_STOP;

END_PROGRAM
```

### Program Logical/main2 (IEC)

#### Main.st
```iecst
PROGRAM _INIT
	// This loop deals with all robot2 control

	// Move to home position
	// If package buffer is not empty, move to above pickup position
	// When sensor.packageForPacker, move down to package height and grab package
	// Move upwards to clear track
	// Move to one of three packing positions
	// Release package
	// ??? Update used position for next package
	// Clear package from buffer
	// Loop end

	// Init robot2
	robot2.state := RSTATE_INIT;
END_PROGRAM

PROGRAM _CYCLIC

	CASE robot2.state OF
		RSTATE_INIT:
			// Set the home position target and wait for arrival
			robot2.target := RTARGET_FORCE_HOME;
			robot2.state := RSTATE_FORCE_HOME;

		RSTATE_FORCE_HOME:
			// Wait for robot to be in position
			IF robot2.inPosition THEN
				// Clear the target IO and wait
				robot2.target := RTARGET_CLEAR;
				robot2.state := RSTATE_WAITING;
			END_IF

		RSTATE_WAITING:
			// Nothing really here

		RSTATE_PICKUP:
			// Sensor loop sent us here, and set a target for us
			// Save this target
			robot2.previousTarget := robot2.target;

			// Wait for robot to be in position
			IF robot2.inPosition THEN
				// Arrived, pick up something
				robot2.grip := TRUE;
				IF robot2.isGripping THEN
					// Gripping, move back to home
					robot2.nextState := RSTATE_PICKUP_R;
					robot2.state := RSTATE_CLEAR;
				END_IF
			END_IF

		RSTATE_PICKUP_R:
			// Select reverse based on previous target
			CASE robot2.previousTarget OF
				RTARGET_PICKUP_1:
					robot2.target := RTARGET_PICKUP_1_R;

				RTARGET_PICKUP_2:
					robot2.target := RTARGET_PICKUP_2_R;

				RTARGET_PICKUP_3:
					robot2.target := RTARGET_PICKUP_3_R;

				RTARGET_PICKUP_4:
					robot2.target := RTARGET_PICKUP_4_R;

			END_CASE

			IF robot2.inPosition THEN
				// If robot says we're home, change to drop state
				robot2.nextState := RSTATE_DROP;
				robot2.state := RSTATE_CLEAR;
			END_IF

		RSTATE_DROP:
			// Select drop target from the first element in the buffer
			CASE packBuffer[0].size OF
				PACKAGE_INVALID:
					// Something is wrong, this should be here ..
					robot2.state := RSTATE_E_STOP;

				PACKAGE_SMALL:
					robot2.target := RTARGET_DROPOFF_1;

				PACKAGE_MEDIUM:
					robot2.target := RTARGET_DROPOFF_2;

				PACKAGE_LARGE:
					robot2.target := RTARGET_DROPOFF_3;

			END_CASE

			// Wait until we're there
			IF robot2.inPosition THEN
				// Save the target
				robot2.previousTarget := robot2.target;

				// Release the package
				robot2.grip := FALSE;
				IF NOT robot2.isGripping THEN
					// State stuff
					robot2.nextState := RSTATE_DROP_R;
					robot2.state := RSTATE_CLEAR;
				END_IF
			END_IF

		RSTATE_DROP_R:
			// Select the path home from previous target
			CASE robot2.previousTarget OF
				RTARGET_DROPOFF_1:
					robot2.target := RTARGET_DROPOFF_1_R;

				RTARGET_DROPOFF_2:
					robot2.target := RTARGET_DROPOFF_2_R;

				RTARGET_DROPOFF_3:
					robot2.target := RTARGET_DROPOFF_3_R;

			END_CASE

			// Wait for inPosition
			IF robot2.inPosition THEN
				// We're ready for new things
				robot2.state := RSTATE_CLEAR;
				robot2.nextState := RSTATE_WAITING;

			END_IF

		RSTATE_CLEAR:
			// Set the state from next set state if filled.
			// We use this to get a cycle of clear IO between moves out and back
			// Else just clear through wait
			IF NOT (robot2.nextState = RSTATE_WAITING) THEN
				robot2.state := robot2.nextState;
				robot2.target := RTARGET_CLEAR;
				robot2.previousTarget := RTARGET_CLEAR;
				robot2.nextState := RSTATE_WAITING;
			ELSE
				robot2.state := RSTATE_WAITING;
			END_IF

		RSTATE_E_STOP:
		// General kill state ..

	END_CASE

	// Write the current IO to robot comm struct, this is ugly AF
	CASE robot2.target OF
		RTARGET_FORCE_HOME:
			robot2.comm.targets.initHome := TRUE;
			robot2.comm.targets.home := FALSE;
			robot2.comm.targets.pick1 := FALSE;
			robot2.comm.targets.pick2 := FALSE;
			robot2.comm.targets.pick3 := FALSE;
			robot2.comm.targets.pick4 := FALSE;
			robot2.comm.targets.drop1 := FALSE;
			robot2.comm.targets.drop2 := FALSE;
			robot2.comm.targets.drop3 := FALSE;

		RTARGET_PICKUP_1:
			robot2.comm.targets.initHome := FALSE;
			robot2.comm.targets.home := FALSE;
			robot2.comm.targets.pick1 := TRUE;
			robot2.comm.targets.pick2 := FALSE;
			robot2.comm.targets.pick3 := FALSE;
			robot2.comm.targets.pick4 := FALSE;
			robot2.comm.targets.drop1 := FALSE;
			robot2.comm.targets.drop2 := FALSE;
			robot2.comm.targets.drop3 := FALSE;
		RTARGET_PICKUP_1_R:
			robot2.comm.targets.initHome := FALSE;
			robot2.comm.targets.home := TRUE;
			robot2.comm.targets.pick1 := TRUE;
			robot2.comm.targets.pick2 := FALSE;
			robot2.comm.targets.pick3 := FALSE;
			robot2.comm.targets.pick4 := FALSE;
			robot2.comm.targets.drop1 := FALSE;
			robot2.comm.targets.drop2 := FALSE;
			robot2.comm.targets.drop3 := FALSE;

		RTARGET_PICKUP_2:
			robot2.comm.targets.initHome := FALSE;
			robot2.comm.targets.home := FALSE;
			robot2.comm.targets.pick1 := FALSE;
			robot2.comm.targets.pick2 := TRUE;
			robot2.comm.targets.pick3 := FALSE;
			robot2.comm.targets.pick4 := FALSE;
			robot2.comm.targets.drop1 := FALSE;
			robot2.comm.targets.drop2 := FALSE;
			robot2.comm.targets.drop3 := FALSE;
		RTARGET_PICKUP_2_R:
			robot2.comm.targets.initHome := FALSE;
			robot2.comm.targets.home := TRUE;
			robot2.comm.targets.pick1 := FALSE;
			robot2.comm.targets.pick2 := TRUE;
			robot2.comm.targets.pick3 := FALSE;
			robot2.comm.targets.pick4 := FALSE;
			robot2.comm.targets.drop1 := FALSE;
			robot2.comm.targets.drop2 := FALSE;
			robot2.comm.targets.drop3 := FALSE;

		RTARGET_PICKUP_3:
			robot2.comm.targets.initHome := FALSE;
			robot2.comm.targets.home := FALSE;
			robot2.comm.targets.pick1 := FALSE;
			robot2.comm.targets.pick2 := FALSE;
			robot2.comm.targets.pick3 := TRUE;
			robot2.comm.targets.pick4 := FALSE;
			robot2.comm.targets.drop1 := FALSE;
			robot2.comm.targets.drop2 := FALSE;
			robot2.comm.targets.drop3 := FALSE;
		RTARGET_PICKUP_3_R:
			robot2.comm.targets.initHome := FALSE;
			robot2.comm.targets.home := TRUE;
			robot2.comm.targets.pick1 := FALSE;
			robot2.comm.targets.pick2 := FALSE;
			robot2.comm.targets.pick3 := TRUE;
			robot2.comm.targets.pick4 := FALSE;
			robot2.comm.targets.drop1 := FALSE;
			robot2.comm.targets.drop2 := FALSE;
			robot2.comm.targets.drop3 := FALSE;

		RTARGET_PICKUP_4:
			robot2.comm.targets.initHome := FALSE;
			robot2.comm.targets.home := FALSE;
			robot2.comm.targets.pick1 := FALSE;
			robot2.comm.targets.pick2 := FALSE;
			robot2.comm.targets.pick3 := FALSE;
			robot2.comm.targets.pick4 := TRUE;
			robot2.comm.targets.drop1 := FALSE;
			robot2.comm.targets.drop2 := FALSE;
			robot2.comm.targets.drop3 := FALSE;
		RTARGET_PICKUP_4_R:
			robot2.comm.targets.initHome := FALSE;
			robot2.comm.targets.home := TRUE;
			robot2.comm.targets.pick1 := FALSE;
			robot2.comm.targets.pick2 := FALSE;
			robot2.comm.targets.pick3 := FALSE;
			robot2.comm.targets.pick4 := TRUE;
			robot2.comm.targets.drop1 := FALSE;
			robot2.comm.targets.drop2 := FALSE;
			robot2.comm.targets.drop3 := FALSE;

		RTARGET_DROPOFF_1:
			robot2.comm.targets.initHome := FALSE;
			robot2.comm.targets.home := FALSE;
			robot2.comm.targets.pick1 := FALSE;
			robot2.comm.targets.pick2 := FALSE;
			robot2.comm.targets.pick3 := FALSE;
			robot2.comm.targets.pick4 := FALSE;
			robot2.comm.targets.drop1 := TRUE;
			robot2.comm.targets.drop2 := FALSE;
			robot2.comm.targets.drop3 := FALSE;
		RTARGET_DROPOFF_1_R:
			robot2.comm.targets.initHome := FALSE;
			robot2.comm.targets.home := TRUE;
			robot2.comm.targets.pick1 := FALSE;
			robot2.comm.targets.pick2 := FALSE;
			robot2.comm.targets.pick3 := FALSE;
			robot2.comm.targets.pick4 := FALSE;
			robot2.comm.targets.drop1 := TRUE;
			robot2.comm.targets.drop2 := FALSE;
			robot2.comm.targets.drop3 := FALSE;

		RTARGET_DROPOFF_2:
			robot2.comm.targets.initHome := FALSE;
			robot2.comm.targets.home := FALSE;
			robot2.comm.targets.pick1 := FALSE;
			robot2.comm.targets.pick2 := FALSE;
			robot2.comm.targets.pick3 := FALSE;
			robot2.comm.targets.pick4 := FALSE;
			robot2.comm.targets.drop1 := FALSE;
			robot2.comm.targets.drop2 := TRUE;
			robot2.comm.targets.drop3 := FALSE;
		RTARGET_DROPOFF_2_R:
			robot2.comm.targets.initHome := FALSE;
			robot2.comm.targets.home := TRUE;
			robot2.comm.targets.pick1 := FALSE;
			robot2.comm.targets.pick2 := FALSE;
			robot2.comm.targets.pick3 := FALSE;
			robot2.comm.targets.pick4 := FALSE;
			robot2.comm.targets.drop1 := FALSE;
			robot2.comm.targets.drop2 := TRUE;
			robot2.comm.targets.drop3 := FALSE;

		RTARGET_DROPOFF_3:
			robot2.comm.targets.initHome := FALSE;
			robot2.comm.targets.home := FALSE;
			robot2.comm.targets.pick1 := FALSE;
			robot2.comm.targets.pick2 := FALSE;
			robot2.comm.targets.pick3 := FALSE;
			robot2.comm.targets.pick4 := FALSE;
			robot2.comm.targets.drop1 := FALSE;
			robot2.comm.targets.drop2 := FALSE;
			robot2.comm.targets.drop3 := TRUE;
		RTARGET_DROPOFF_3_R:
			robot2.comm.targets.initHome := FALSE;
			robot2.comm.targets.home := TRUE;
			robot2.comm.targets.pick1 := FALSE;
			robot2.comm.targets.pick2 := FALSE;
			robot2.comm.targets.pick3 := FALSE;
			robot2.comm.targets.pick4 := FALSE;
			robot2.comm.targets.drop1 := FALSE;
			robot2.comm.targets.drop2 := FALSE;
			robot2.comm.targets.drop3 := TRUE;

		RTARGET_CLEAR:
			robot2.comm.targets.initHome := FALSE;
			robot2.comm.targets.home := FALSE;
			robot2.comm.targets.pick1 := FALSE;
			robot2.comm.targets.pick2 := FALSE;
			robot2.comm.targets.pick3 := FALSE;
			robot2.comm.targets.pick4 := FALSE;
			robot2.comm.targets.drop1 := FALSE;
			robot2.comm.targets.drop2 := FALSE;
			robot2.comm.targets.drop3 := FALSE;

	END_CASE
	robot2.comm.doGrip := robot2.grip;
	robot2.isGripping := robot2.comm.diGrip;
	robot2.inPosition := robot2.comm.inPosition;
	robot2.isWaiting := robot2.comm.isWaiting;

END_PROGRAM

PROGRAM _EXIT
	(* Insert code here *)

END_PROGRAM
```

Listed in the project but not available here: Logical/Libraries
